(* CoDeSys 2.3 library: Visu_Scheduler_03_e.lib *)
(* Libraries: Standard.lib 4.10.05 11:14:46, SYSLIBCALLBACK.LIB*7.9.10 14:37:47 *)

(* POU Fu_Version_Visu_Scheduler, ST *)
FUNCTION Fu_Version_Visu_Scheduler : WORD
(*******************************************************************************
  WAGO Kontakttechnik GmbH Hansastr. 27 32423 Minden(Westf.) 
  Tel. +49571/887-0                                                                                                
   
  Function	: This function ist for checking purposes of the version.
 
  Version	: 3.1
  Date		: 14.03.2011

*******************************************************************************)
VAR_INPUT
	EN : BOOL;
END_VAR
Fu_Version_Visu_Scheduler:=16#0301;
(*
***** 26.01.2011, V3.0 *****************************************************
 - Release of the library Scheduler_03.lib and Visu_Scheduler_03.lib

***** 14.03.2011, V3.1*****************************************************
 - visuTimetable_e: Adjust the Input field for individual end time on Friday
*)
END_FUNCTION

(* Visualisation visuHoliday
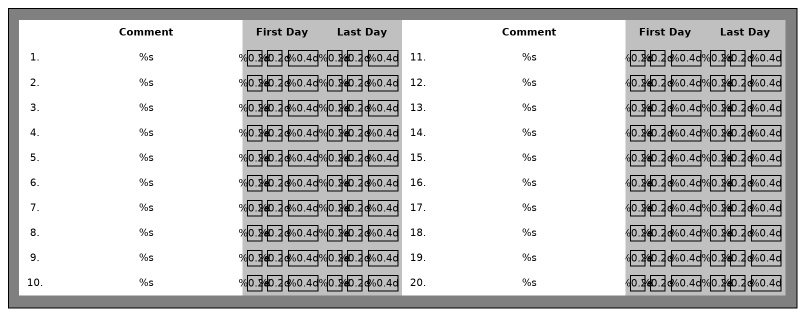
rectangle at (234,36)-(314,62): text "-     -"; tooltip First day Input format: DD-HH-YYYY
rectangle at (314,36)-(394,62): text "-     -"; tooltip Last day Input format: DD-HH-YYYY
rectangle at (319,42)-(334,58): text "%0.2d"; shows $typHoliday$.wLastDay[1,1]; editable 0..31
rectangle at (339,42)-(354,58): text "%0.2d"; shows $typHoliday$.wLastDay[2,1]; editable 0..12
rectangle at (360,42)-(390,58): text "%0.4d"; shows $typHoliday$.wLastDay[3,1]; editable 0..2099
rectangle at (43,36)-(234,62): text "%s"; shows $typHoliday$.strComment[1]; editable
rectangle at (234,62)-(314,87): text "-     -"; tooltip First day Input format: DD-HH-YYYY
rectangle at (314,62)-(394,87): text "-     -"; tooltip Last day Input format: DD-HH-YYYY
rectangle at (319,67)-(334,83): text "%0.2d"; shows $typHoliday$.wLastDay[1,2]; editable 0..31
rectangle at (339,67)-(354,83): text "%0.2d"; shows $typHoliday$.wLastDay[2,2]; editable 0..12
rectangle at (360,67)-(390,83): text "%0.4d"; shows $typHoliday$.wLastDay[3,2]; editable 0..2099
rectangle at (43,62)-(234,87): text "%s"; shows $typHoliday$.strComment[2]; editable
rectangle at (234,87)-(314,112): text "-     -"; tooltip First day Input format: DD-HH-YYYY
rectangle at (314,87)-(394,112): text "-     -"; tooltip Last day Input format: DD-HH-YYYY
rectangle at (319,92)-(334,108): text "%0.2d"; shows $typHoliday$.wLastDay[1,3]; editable 0..31
rectangle at (339,92)-(354,108): text "%0.2d"; shows $typHoliday$.wLastDay[2,3]; editable 0..12
rectangle at (360,92)-(390,108): text "%0.4d"; shows $typHoliday$.wLastDay[3,3]; editable 0..2099
rectangle at (43,87)-(234,112): text "%s"; shows $typHoliday$.strComment[3]; editable
rectangle at (234,112)-(314,137): text "-     -"; tooltip First day Input format: DD-HH-YYYY
rectangle at (314,112)-(394,137): text "-     -"; tooltip Last day Input format: DD-HH-YYYY
rectangle at (319,117)-(334,133): text "%0.2d"; shows $typHoliday$.wLastDay[1,4]; editable 0..31
rectangle at (339,117)-(354,133): text "%0.2d"; shows $typHoliday$.wLastDay[2,4]; editable 0..12
rectangle at (360,117)-(390,133): text "%0.4d"; shows $typHoliday$.wLastDay[3,4]; editable 0..2099
rectangle at (43,112)-(234,137): text "%s"; shows $typHoliday$.strComment[4]; editable
rectangle at (234,137)-(314,162): text "-     -"; tooltip First day Input format: DD-HH-YYYY
rectangle at (314,137)-(394,162): text "-     -"; tooltip Last day Input format: DD-HH-YYYY
rectangle at (319,142)-(334,158): text "%0.2d"; shows $typHoliday$.wLastDay[1,5]; editable 0..31
rectangle at (339,142)-(354,158): text "%0.2d"; shows $typHoliday$.wLastDay[2,5]; editable 0..12
rectangle at (360,142)-(390,158): text "%0.4d"; shows $typHoliday$.wLastDay[3,5]; editable 0..2099
rectangle at (43,137)-(234,162): text "%s"; shows $typHoliday$.strComment[5]; editable
rectangle at (234,162)-(314,187): text "-     -"; tooltip First day Input format: DD-HH-YYYY
rectangle at (314,162)-(394,187): text "-     -"; tooltip Last day Input format: DD-HH-YYYY
rectangle at (319,167)-(334,183): text "%0.2d"; shows $typHoliday$.wLastDay[1,6]; editable 0..31
rectangle at (339,167)-(354,183): text "%0.2d"; shows $typHoliday$.wLastDay[2,6]; editable 0..12
rectangle at (360,167)-(390,183): text "%0.4d"; shows $typHoliday$.wLastDay[3,6]; editable 0..2099
rectangle at (43,162)-(234,187): text "%s"; shows $typHoliday$.strComment[6]; editable
rectangle at (234,187)-(314,212): text "-     -"; tooltip First day Input format: DD-HH-YYYY
rectangle at (314,187)-(394,212): text "-     -"; tooltip Last day Input format: DD-HH-YYYY
rectangle at (319,192)-(334,208): text "%0.2d"; shows $typHoliday$.wLastDay[1,7]; editable 0..31
rectangle at (339,192)-(354,208): text "%0.2d"; shows $typHoliday$.wLastDay[2,7]; editable 0..12
rectangle at (360,192)-(390,208): text "%0.4d"; shows $typHoliday$.wLastDay[3,7]; editable 0..2099
rectangle at (43,187)-(234,212): text "%s"; shows $typHoliday$.strComment[7]; editable
rectangle at (234,212)-(314,237): text "-     -"; tooltip First day Input format: DD-HH-YYYY
rectangle at (314,212)-(394,237): text "-     -"; tooltip Last day Input format: DD-HH-YYYY
rectangle at (319,217)-(334,233): text "%0.2d"; shows $typHoliday$.wLastDay[1,8]; editable 0..31
rectangle at (339,217)-(354,233): text "%0.2d"; shows $typHoliday$.wLastDay[2,8]; editable 0..12
rectangle at (360,217)-(390,233): text "%0.4d"; shows $typHoliday$.wLastDay[3,8]; editable 0..2099
rectangle at (43,212)-(234,237): text "%s"; shows $typHoliday$.strComment[8]; editable
rectangle at (234,237)-(314,262): text "-     -"; tooltip First day Input format: DD-HH-YYYY
rectangle at (314,237)-(394,262): text "-     -"; tooltip Last day Input format: DD-HH-YYYY
rectangle at (319,242)-(334,258): text "%0.2d"; shows $typHoliday$.wLastDay[1,9]; editable 0..31
rectangle at (339,242)-(354,258): text "%0.2d"; shows $typHoliday$.wLastDay[2,9]; editable 0..12
rectangle at (360,242)-(390,258): text "%0.4d"; shows $typHoliday$.wLastDay[3,9]; editable 0..2099
rectangle at (43,237)-(234,262): text "%s"; shows $typHoliday$.strComment[9]; editable
rectangle at (234,262)-(314,287): text "-     -"; tooltip First day Input format: DD-HH-YYYY
rectangle at (314,262)-(394,287): text "-     -"; tooltip Last day Input format: DD-HH-YYYY
rectangle at (319,267)-(334,283): text "%0.2d"; shows $typHoliday$.wLastDay[1,10]; editable 0..31
rectangle at (339,267)-(354,283): text "%0.2d"; shows $typHoliday$.wLastDay[2,10]; editable 0..12
rectangle at (360,267)-(390,283): text "%0.4d"; shows $typHoliday$.wLastDay[3,10]; editable 0..2099
rectangle at (43,262)-(234,287): text "%s"; shows $typHoliday$.strComment[10]; editable
rectangle at (617,36)-(697,62): text "-     -"; tooltip First day Input format: DD-HH-YYYY
rectangle at (622,42)-(637,58): text "%0.2d"; shows $typHoliday$.wFirstDay[1,11]; editable 0..31
rectangle at (642,42)-(657,58): text "%0.2d"; shows $typHoliday$.wFirstDay[2,11]; editable 0..12
rectangle at (663,42)-(693,58): text "%0.4d"; shows $typHoliday$.wFirstDay[3,11]; editable 0..2099
rectangle at (697,36)-(777,62): text "-     -"; tooltip Last day Input format: DD-HH-YYYY
rectangle at (702,42)-(717,58): text "%0.2d"; shows $typHoliday$.wLastDay[1,11]; editable 0..31
rectangle at (722,42)-(737,58): text "%0.2d"; shows $typHoliday$.wLastDay[2,11]; editable 0..12
rectangle at (743,42)-(773,58): text "%0.4d"; shows $typHoliday$.wLastDay[3,11]; editable 0..2099
rectangle at (426,36)-(617,62): text "%s"; shows $typHoliday$.strComment[11]; editable
rectangle at (617,62)-(697,87): text "-     -"; tooltip First day Input format: DD-HH-YYYY
rectangle at (622,67)-(637,83): text "%0.2d"; shows $typHoliday$.wFirstDay[1,12]; editable 0..31
rectangle at (642,67)-(657,83): text "%0.2d"; shows $typHoliday$.wFirstDay[2,12]; editable 0..12
rectangle at (663,67)-(693,83): text "%0.4d"; shows $typHoliday$.wFirstDay[3,12]; editable 0..2099
rectangle at (697,62)-(777,87): text "-     -"; tooltip Last day Input format: DD-HH-YYYY
rectangle at (702,67)-(717,83): text "%0.2d"; shows $typHoliday$.wLastDay[1,12]; editable 0..31
rectangle at (722,67)-(737,83): text "%0.2d"; shows $typHoliday$.wLastDay[2,12]; editable 0..12
rectangle at (743,67)-(773,83): text "%0.4d"; shows $typHoliday$.wLastDay[3,12]; editable 0..2099
rectangle at (426,62)-(617,87): text "%s"; shows $typHoliday$.strComment[12]; editable
rectangle at (617,87)-(697,112): text "-     -"; tooltip First day Input format: DD-HH-YYYY
rectangle at (622,92)-(637,108): text "%0.2d"; shows $typHoliday$.wFirstDay[1,13]; editable 0..31
rectangle at (642,92)-(657,108): text "%0.2d"; shows $typHoliday$.wFirstDay[2,13]; editable 0..12
rectangle at (663,92)-(693,108): text "%0.4d"; shows $typHoliday$.wFirstDay[3,13]; editable 0..2099
rectangle at (697,87)-(777,112): text "-     -"; tooltip Last day Input format: DD-HH-YYYY
rectangle at (702,92)-(717,108): text "%0.2d"; shows $typHoliday$.wLastDay[1,13]; editable 0..31
rectangle at (722,92)-(737,108): text "%0.2d"; shows $typHoliday$.wLastDay[2,13]; editable 0..12
rectangle at (743,92)-(773,108): text "%0.4d"; shows $typHoliday$.wLastDay[3,13]; editable 0..2099
rectangle at (426,87)-(617,112): text "%s"; shows $typHoliday$.strComment[13]; editable
rectangle at (617,112)-(697,137): text "-     -"; tooltip First day Input format: DD-HH-YYYY
rectangle at (622,117)-(637,133): text "%0.2d"; shows $typHoliday$.wFirstDay[1,14]; editable 0..31
rectangle at (642,117)-(657,133): text "%0.2d"; shows $typHoliday$.wFirstDay[2,14]; editable 0..12
rectangle at (663,117)-(693,133): text "%0.4d"; shows $typHoliday$.wFirstDay[3,14]; editable 0..2099
rectangle at (697,112)-(777,137): text "-     -"; tooltip Last day Input format: DD-HH-YYYY
rectangle at (702,117)-(717,133): text "%0.2d"; shows $typHoliday$.wLastDay[1,14]; editable 0..31
rectangle at (722,117)-(737,133): text "%0.2d"; shows $typHoliday$.wLastDay[2,14]; editable 0..12
rectangle at (743,117)-(773,133): text "%0.4d"; shows $typHoliday$.wLastDay[3,14]; editable 0..2099
rectangle at (426,112)-(617,137): text "%s"; shows $typHoliday$.strComment[14]; editable
rectangle at (617,137)-(697,162): text "-     -"; tooltip First day Input format: DD-HH-YYYY
rectangle at (622,142)-(637,158): text "%0.2d"; shows $typHoliday$.wFirstDay[1,15]; editable 0..31
rectangle at (642,142)-(657,158): text "%0.2d"; shows $typHoliday$.wFirstDay[2,15]; editable 0..12
rectangle at (663,142)-(693,158): text "%0.4d"; shows $typHoliday$.wFirstDay[3,15]; editable 0..2099
rectangle at (697,137)-(777,162): text "-     -"; tooltip Last day Input format: DD-HH-YYYY
rectangle at (702,142)-(717,158): text "%0.2d"; shows $typHoliday$.wLastDay[1,15]; editable 0..31
rectangle at (722,142)-(737,158): text "%0.2d"; shows $typHoliday$.wLastDay[2,15]; editable 0..12
rectangle at (743,142)-(773,158): text "%0.4d"; shows $typHoliday$.wLastDay[3,15]; editable 0..2099
rectangle at (426,137)-(617,162): text "%s"; shows $typHoliday$.strComment[15]; editable
rectangle at (617,162)-(697,187): text "-     -"; tooltip First day Input format: DD-HH-YYYY
rectangle at (622,167)-(637,183): text "%0.2d"; shows $typHoliday$.wFirstDay[1,16]; editable 0..31
rectangle at (642,167)-(657,183): text "%0.2d"; shows $typHoliday$.wFirstDay[2,16]; editable 0..12
rectangle at (663,167)-(693,183): text "%0.4d"; shows $typHoliday$.wFirstDay[3,16]; editable 0..2099
rectangle at (697,162)-(777,187): text "-     -"; tooltip Last day Input format: DD-HH-YYYY
rectangle at (702,167)-(717,183): text "%0.2d"; shows $typHoliday$.wLastDay[1,16]; editable 0..31
rectangle at (722,167)-(737,183): text "%0.2d"; shows $typHoliday$.wLastDay[2,16]; editable 0..12
rectangle at (743,167)-(773,183): text "%0.4d"; shows $typHoliday$.wLastDay[3,16]; editable 0..2099
rectangle at (426,162)-(617,187): text "%s"; shows $typHoliday$.strComment[16]; editable
rectangle at (617,187)-(697,212): text "-     -"; tooltip First day Input format: DD-HH-YYYY
rectangle at (622,192)-(637,208): text "%0.2d"; shows $typHoliday$.wFirstDay[1,17]; editable 0..31
rectangle at (642,192)-(657,208): text "%0.2d"; shows $typHoliday$.wFirstDay[2,17]; editable 0..12
rectangle at (663,192)-(693,208): text "%0.4d"; shows $typHoliday$.wFirstDay[3,17]; editable 0..2099
rectangle at (697,187)-(777,212): text "-     -"; tooltip Last day Input format: DD-HH-YYYY
rectangle at (702,192)-(717,208): text "%0.2d"; shows $typHoliday$.wLastDay[1,17]; editable 0..31
rectangle at (722,192)-(737,208): text "%0.2d"; shows $typHoliday$.wLastDay[2,17]; editable 0..12
rectangle at (743,192)-(773,208): text "%0.4d"; shows $typHoliday$.wLastDay[3,17]; editable 0..2099
rectangle at (426,187)-(617,212): text "%s"; shows $typHoliday$.strComment[17]; editable
rectangle at (617,212)-(697,237): text "-     -"; tooltip First day Input format: DD-HH-YYYY
rectangle at (622,217)-(637,233): text "%0.2d"; shows $typHoliday$.wFirstDay[1,18]; editable 0..31
rectangle at (642,217)-(657,233): text "%0.2d"; shows $typHoliday$.wFirstDay[2,18]; editable 0..12
rectangle at (663,217)-(693,233): text "%0.4d"; shows $typHoliday$.wFirstDay[3,18]; editable 0..2099
rectangle at (697,212)-(777,237): text "-     -"; tooltip Last day Input format: DD-HH-YYYY
rectangle at (702,217)-(717,233): text "%0.2d"; shows $typHoliday$.wLastDay[1,18]; editable 0..31
rectangle at (722,217)-(737,233): text "%0.2d"; shows $typHoliday$.wLastDay[2,18]; editable 0..12
rectangle at (743,217)-(773,233): text "%0.4d"; shows $typHoliday$.wLastDay[3,18]; editable 0..2099
rectangle at (426,212)-(617,237): text "%s"; shows $typHoliday$.strComment[18]; editable
rectangle at (617,237)-(697,262): text "-     -"; tooltip First day Input format: DD-HH-YYYY
rectangle at (622,242)-(637,258): text "%0.2d"; shows $typHoliday$.wFirstDay[1,19]; editable 0..31
rectangle at (642,242)-(657,258): text "%0.2d"; shows $typHoliday$.wFirstDay[2,19]; editable 0..12
rectangle at (663,242)-(693,258): text "%0.4d"; shows $typHoliday$.wFirstDay[3,19]; editable 0..2099
rectangle at (697,237)-(777,262): text "-     -"; tooltip Last day Input format: DD-HH-YYYY
rectangle at (702,242)-(717,258): text "%0.2d"; shows $typHoliday$.wLastDay[1,19]; editable 0..31
rectangle at (722,242)-(737,258): text "%0.2d"; shows $typHoliday$.wLastDay[2,19]; editable 0..12
rectangle at (743,242)-(773,258): text "%0.4d"; shows $typHoliday$.wLastDay[3,19]; editable 0..2099
rectangle at (426,237)-(617,262): text "%s"; shows $typHoliday$.strComment[19]; editable
rectangle at (617,262)-(697,287): text "-     -"; tooltip First day Input format: DD-HH-YYYY
rectangle at (622,267)-(637,283): text "%0.2d"; shows $typHoliday$.wFirstDay[1,20]; editable 0..31
rectangle at (642,267)-(657,283): text "%0.2d"; shows $typHoliday$.wFirstDay[2,20]; editable 0..12
rectangle at (663,267)-(693,283): text "%0.4d"; shows $typHoliday$.wFirstDay[3,20]; editable 0..2099
rectangle at (697,262)-(777,287): text "-     -"; tooltip Last day Input format: DD-HH-YYYY
rectangle at (702,267)-(717,283): text "%0.2d"; shows $typHoliday$.wLastDay[1,20]; editable 0..31
rectangle at (722,267)-(737,283): text "%0.2d"; shows $typHoliday$.wLastDay[2,20]; editable 0..12
rectangle at (743,267)-(773,283): text "%0.4d"; shows $typHoliday$.wLastDay[3,20]; editable 0..2099
rectangle at (426,262)-(617,287): text "%s"; shows $typHoliday$.strComment[20]; editable
rectangle at (11,36)-(43,62): text "1."
rectangle at (11,62)-(43,87): text "2."
rectangle at (11,87)-(43,112): text "3."
rectangle at (11,112)-(43,137): text "4."
rectangle at (11,137)-(43,162): text "5."
rectangle at (11,162)-(43,187): text "6."
rectangle at (11,187)-(43,212): text "7."
rectangle at (11,212)-(43,237): text "8."
rectangle at (11,237)-(43,262): text "9."
rectangle at (11,262)-(43,287): text "10."
rectangle at (394,36)-(426,62): text "11."
rectangle at (394,62)-(426,87): text "12."
rectangle at (394,87)-(426,112): text "13."
rectangle at (394,112)-(426,137): text "14."
rectangle at (394,137)-(426,162): text "15."
rectangle at (394,162)-(426,187): text "16."
rectangle at (394,187)-(426,212): text "17."
rectangle at (394,212)-(426,237): text "18."
rectangle at (394,237)-(426,262): text "19."
rectangle at (394,262)-(426,287): text "20."
rectangle at (617,12)-(697,36): text "First Day"
rectangle at (697,12)-(777,36): text "Last Day"
rectangle at (426,12)-(617,36): text "Comment"
rectangle at (234,12)-(314,36): text "First Day"
rectangle at (314,12)-(394,36): text "Last Day"
rectangle at (43,12)-(234,36): text "Comment"
rectangle at (239,42)-(254,58): text "%0.2d"; shows $typHoliday$.wFirstDay[1,1]; editable 0..31
rectangle at (259,42)-(274,58): text "%0.2d"; shows $typHoliday$.wFirstDay[2,1]; editable 0..12
rectangle at (280,42)-(310,58): text "%0.4d"; shows $typHoliday$.wFirstDay[3,1]; editable 0..2099
rectangle at (239,67)-(254,83): text "%0.2d"; shows $typHoliday$.wFirstDay[1,2]; editable 0..31
rectangle at (259,67)-(274,83): text "%0.2d"; shows $typHoliday$.wFirstDay[2,2]; editable 0..12
rectangle at (280,67)-(310,83): text "%0.4d"; shows $typHoliday$.wFirstDay[3,2]; editable 0..2099
rectangle at (239,92)-(254,108): text "%0.2d"; shows $typHoliday$.wFirstDay[1,3]; editable 0..31
rectangle at (259,92)-(274,108): text "%0.2d"; shows $typHoliday$.wFirstDay[2,3]; editable 0..12
rectangle at (280,92)-(310,108): text "%0.4d"; shows $typHoliday$.wFirstDay[3,3]; editable 0..2099
rectangle at (239,117)-(254,133): text "%0.2d"; shows $typHoliday$.wFirstDay[1,4]; editable 0..31
rectangle at (259,117)-(274,133): text "%0.2d"; shows $typHoliday$.wFirstDay[2,4]; editable 0..12
rectangle at (280,117)-(310,133): text "%0.4d"; shows $typHoliday$.wFirstDay[3,4]; editable 0..2099
rectangle at (239,142)-(254,158): text "%0.2d"; shows $typHoliday$.wFirstDay[1,5]; editable 0..31
rectangle at (259,142)-(274,158): text "%0.2d"; shows $typHoliday$.wFirstDay[2,5]; editable 0..12
rectangle at (280,142)-(310,158): text "%0.4d"; shows $typHoliday$.wFirstDay[3,5]; editable 0..2099
rectangle at (239,167)-(254,183): text "%0.2d"; shows $typHoliday$.wFirstDay[1,6]; editable 0..31
rectangle at (259,167)-(274,183): text "%0.2d"; shows $typHoliday$.wFirstDay[2,6]; editable 0..12
rectangle at (280,167)-(310,183): text "%0.4d"; shows $typHoliday$.wFirstDay[3,6]; editable 0..2099
rectangle at (239,192)-(254,208): text "%0.2d"; shows $typHoliday$.wFirstDay[1,7]; editable 0..31
rectangle at (259,192)-(274,208): text "%0.2d"; shows $typHoliday$.wFirstDay[2,7]; editable 0..12
rectangle at (280,192)-(310,208): text "%0.4d"; shows $typHoliday$.wFirstDay[3,7]; editable 0..2099
rectangle at (239,217)-(254,233): text "%0.2d"; shows $typHoliday$.wFirstDay[1,8]; editable 0..31
rectangle at (259,217)-(274,233): text "%0.2d"; shows $typHoliday$.wFirstDay[2,8]; editable 0..12
rectangle at (280,217)-(310,233): text "%0.4d"; shows $typHoliday$.wFirstDay[3,8]; editable 0..2099
rectangle at (239,242)-(254,258): text "%0.2d"; shows $typHoliday$.wFirstDay[1,9]; editable 0..31
rectangle at (259,242)-(274,258): text "%0.2d"; shows $typHoliday$.wFirstDay[2,9]; editable 0..12
rectangle at (280,242)-(310,258): text "%0.4d"; shows $typHoliday$.wFirstDay[3,9]; editable 0..2099
rectangle at (239,267)-(254,283): text "%0.2d"; shows $typHoliday$.wFirstDay[1,10]; editable 0..31
rectangle at (259,267)-(274,283): text "%0.2d"; shows $typHoliday$.wFirstDay[2,10]; editable 0..12
rectangle at (280,267)-(310,283): text "%0.4d"; shows $typHoliday$.wFirstDay[3,10]; editable 0..2099
5 more shapes without text or variables
*)

(* Visualisation visuPublicHoliday
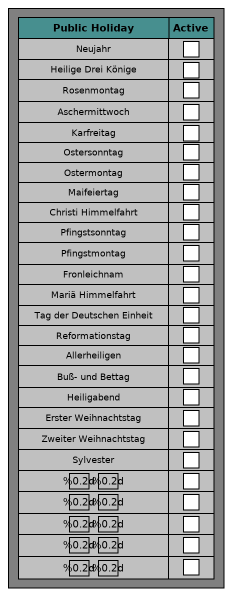
rectangle at (160,9)-(206,31): text "Active"
rectangle at (10,9)-(161,31): text "Public Holiday"
rectangle at (10,30)-(161,52): text "Neujahr"
rectangle at (175,33)-(191,49): alarm colour if $typPublicHoliday$.Neujahr; toggles $typPublicHoliday$.Neujahr; tooltip Wenn dieses Feld aktiviert ist, wird der Feiertag für die Feiertagserkennung im "FbPublicHoliday" berücksichtigt.
rectangle at (10,51)-(161,72): text "Heilige Drei Könige"
rectangle at (175,54)-(191,70): alarm colour if $typPublicHoliday$.Heilige_Drei_Koenige; toggles $typPublicHoliday$.Heilige_Drei_Koenige; tooltip Wenn dieses Feld aktiviert ist, wird der Feiertag für die Feiertagserkennung im "FbPublicHoliday" berücksichtigt.
rectangle at (10,71)-(161,94): text "Rosenmontag"
rectangle at (175,74)-(191,90): alarm colour if $typPublicHoliday$.Rosenmontag; toggles $typPublicHoliday$.Rosenmontag; tooltip Wenn dieses Feld aktiviert ist, wird der Feiertag für die Feiertagserkennung im "FbPublicHoliday" berücksichtigt.
rectangle at (10,93)-(161,115): text "Aschermittwoch"
rectangle at (175,96)-(191,112): alarm colour if $typPublicHoliday$.Aschermittwoch; toggles $typPublicHoliday$.Aschermittwoch; tooltip Wenn dieses Feld aktiviert ist, wird der Feiertag für die Feiertagserkennung im "FbPublicHoliday" berücksichtigt.
rectangle at (10,114)-(161,136): text "Karfreitag"
rectangle at (175,117)-(191,133): alarm colour if $typPublicHoliday$.Karfreitag; toggles $typPublicHoliday$.Karfreitag; tooltip Wenn dieses Feld aktiviert ist, wird der Feiertag für die Feiertagserkennung im "FbPublicHoliday" berücksichtigt.
rectangle at (10,134)-(161,155): text "Ostersonntag"
rectangle at (175,136)-(191,152): alarm colour if $typPublicHoliday$.Ostersonntag; toggles $typPublicHoliday$.Ostersonntag; tooltip Wenn dieses Feld aktiviert ist, wird der Feiertag für die Feiertagserkennung im "FbPublicHoliday" berücksichtigt.
rectangle at (10,154)-(161,176): text "Ostermontag"
rectangle at (175,156)-(191,172): alarm colour if $typPublicHoliday$.Ostermontag; toggles $typPublicHoliday$.Ostermontag; tooltip Wenn dieses Feld aktiviert ist, wird der Feiertag für die Feiertagserkennung im "FbPublicHoliday" berücksichtigt.
rectangle at (10,174)-(161,195): text "Maifeiertag"
rectangle at (175,176)-(191,192): alarm colour if $typPublicHoliday$.Maifeiertag; toggles $typPublicHoliday$.Maifeiertag; tooltip Wenn dieses Feld aktiviert ist, wird der Feiertag für die Feiertagserkennung im "FbPublicHoliday" berücksichtigt.
rectangle at (10,194)-(161,215): text "Christi Himmelfahrt"
rectangle at (175,196)-(191,212): alarm colour if $typPublicHoliday$.Christi_Himmelfahrt; toggles $typPublicHoliday$.Christi_Himmelfahrt; tooltip Wenn dieses Feld aktiviert ist, wird der Feiertag für die Feiertagserkennung im "FbPublicHoliday" berücksichtigt.
rectangle at (10,214)-(161,235): text "Pfingstsonntag"
rectangle at (175,216)-(191,232): alarm colour if $typPublicHoliday$.Pfingstsonntag; toggles $typPublicHoliday$.Pfingstsonntag; tooltip Wenn dieses Feld aktiviert ist, wird der Feiertag für die Feiertagserkennung im "FbPublicHoliday" berücksichtigt.
rectangle at (10,234)-(161,257): text "Pfingstmontag"
rectangle at (175,237)-(191,253): alarm colour if $typPublicHoliday$.Pfingstmontag; toggles $typPublicHoliday$.Pfingstmontag; tooltip Wenn dieses Feld aktiviert ist, wird der Feiertag für die Feiertagserkennung im "FbPublicHoliday" berücksichtigt.
rectangle at (10,256)-(161,277): text "Fronleichnam"
rectangle at (175,258)-(191,274): alarm colour if $typPublicHoliday$.Fronleichnam; toggles $typPublicHoliday$.Fronleichnam; tooltip Wenn dieses Feld aktiviert ist, wird der Feiertag für die Feiertagserkennung im "FbPublicHoliday" berücksichtigt.
rectangle at (10,276)-(161,298): text "Mariä Himmelfahrt"
rectangle at (175,279)-(191,295): alarm colour if $typPublicHoliday$.Mariae_Himmelfahrt; toggles $typPublicHoliday$.Mariae_Himmelfahrt; tooltip Wenn dieses Feld aktiviert ist, wird der Feiertag für die Feiertagserkennung im "FbPublicHoliday" berücksichtigt.
rectangle at (10,297)-(161,318): text "Tag der Deutschen Einheit"
rectangle at (175,299)-(191,315): alarm colour if $typPublicHoliday$.Tag_der_Deutschen_Einheit; toggles $typPublicHoliday$.Tag_der_Deutschen_Einheit; tooltip Wenn dieses Feld aktiviert ist, wird der Feiertag für die Feiertagserkennung im "FbPublicHoliday" berücksichtigt.
rectangle at (10,317)-(161,339): text "Reformationstag"
rectangle at (175,319)-(191,335): alarm colour if $typPublicHoliday$.Reformationstag; toggles $typPublicHoliday$.Reformationstag; tooltip Wenn dieses Feld aktiviert ist, wird der Feiertag für die Feiertagserkennung im "FbPublicHoliday" berücksichtigt.
rectangle at (10,337)-(161,358): text "Allerheiligen"
rectangle at (175,339)-(191,355): alarm colour if $typPublicHoliday$.Allerheiligen; toggles $typPublicHoliday$.Allerheiligen; tooltip Wenn dieses Feld aktiviert ist, wird der Feiertag für die Feiertagserkennung im "FbPublicHoliday" berücksichtigt.
rectangle at (10,357)-(161,381): text "Buß- und Bettag"
rectangle at (175,360)-(191,376): alarm colour if $typPublicHoliday$.Buss_und_Bettag; toggles $typPublicHoliday$.Buss_und_Bettag; tooltip Wenn dieses Feld aktiviert ist, wird der Feiertag für die Feiertagserkennung im "FbPublicHoliday" berücksichtigt.
rectangle at (10,379)-(161,400): text "Heiligabend"
rectangle at (175,381)-(191,397): alarm colour if $typPublicHoliday$.Heiligabend; toggles $typPublicHoliday$.Heiligabend; tooltip Wenn dieses Feld aktiviert ist, wird der Feiertag für die Feiertagserkennung im "FbPublicHoliday" berücksichtigt.
rectangle at (10,399)-(161,421): text "Erster Weihnachtstag"
rectangle at (175,402)-(191,418): alarm colour if $typPublicHoliday$.Erster_Weihnachtstag; toggles $typPublicHoliday$.Erster_Weihnachtstag; tooltip Wenn dieses Feld aktiviert ist, wird der Feiertag für die Feiertagserkennung im "FbPublicHoliday" berücksichtigt.
rectangle at (10,420)-(161,442): text "Zweiter Weihnachtstag"
rectangle at (175,423)-(191,439): alarm colour if $typPublicHoliday$.Zweiter_Weihnachtstag; toggles $typPublicHoliday$.Zweiter_Weihnachtstag; tooltip Wenn dieses Feld aktiviert ist, wird der Feiertag für die Feiertagserkennung im "FbPublicHoliday" berücksichtigt.
rectangle at (10,441)-(161,463): text "Sylvester"
rectangle at (175,444)-(191,460): alarm colour if $typPublicHoliday$.Sylvester; toggles $typPublicHoliday$.Sylvester; tooltip Wenn dieses Feld aktiviert ist, wird der Feiertag für die Feiertagserkennung im "FbPublicHoliday" berücksichtigt.
rectangle at (10,462)-(161,485): text "-"; tooltip Eingabeformat:DD-MM Es können beliebige Feiertage mit ihrem Datum vorgegeben werden.
rectangle at (175,465)-(191,481): alarm colour if $typPublicHoliday$.SetSpecialPublicHoliday.0; toggles $typPublicHoliday$.SetSpecialPublicHoliday.0; tooltip Wenn dieses Feld aktiviert ist, wird der Feiertag für die Feiertagserkennung im "FbPublicHoliday" berücksichtigt.
rectangle at (10,483)-(161,506): text "-"; tooltip Eingabeformat:DD-MM Es können beliebige Feiertage mit ihrem Datum vorgegeben werden.
rectangle at (10,505)-(161,528): text "-"; tooltip Eingabeformat:DD-MM Es können beliebige Feiertage mit ihrem Datum vorgegeben werden.
rectangle at (10,526)-(161,549): text "-"; tooltip Eingabeformat:DD-MM Es können beliebige Feiertage mit ihrem Datum vorgegeben werden.
rectangle at (10,548)-(161,571): text "-"; tooltip Eingabeformat:DD-MM Es können beliebige Feiertage mit ihrem Datum vorgegeben werden.
rectangle at (175,486)-(191,502): alarm colour if $typPublicHoliday$.SetSpecialPublicHoliday.1; toggles $typPublicHoliday$.SetSpecialPublicHoliday.1; tooltip Wenn dieses Feld aktiviert ist, wird der Feiertag für die Feiertagserkennung im "FbPublicHoliday" berücksichtigt.
rectangle at (175,508)-(191,524): alarm colour if $typPublicHoliday$.SetSpecialPublicHoliday.2; toggles $typPublicHoliday$.SetSpecialPublicHoliday.2; tooltip Wenn dieses Feld aktiviert ist, wird der Feiertag für die Feiertagserkennung im "FbPublicHoliday" berücksichtigt.
rectangle at (175,529)-(191,545): alarm colour if $typPublicHoliday$.SetSpecialPublicHoliday.3; toggles $typPublicHoliday$.SetSpecialPublicHoliday.3; tooltip Wenn dieses Feld aktiviert ist, wird der Feiertag für die Feiertagserkennung im "FbPublicHoliday" berücksichtigt.
rectangle at (175,551)-(191,567): alarm colour if $typPublicHoliday$.SetSpecialPublicHoliday.4; toggles $typPublicHoliday$.SetSpecialPublicHoliday.4; tooltip Wenn dieses Feld aktiviert ist, wird der Feiertag für die Feiertagserkennung im "FbPublicHoliday" berücksichtigt.
rectangle at (90,465)-(110,481): text "%0.2d"; shows $typPublicHoliday$.SpecialPublicHoliday1_month; editable 1..12
rectangle at (61,465)-(81,481): text "%0.2d"; shows $typPublicHoliday$.SpecialPublicHoliday1_day; editable 1..31
rectangle at (90,486)-(110,502): text "%0.2d"; shows $typPublicHoliday$.SpecialPublicHoliday2_month; editable 1..12
rectangle at (61,486)-(81,502): text "%0.2d"; shows $typPublicHoliday$.SpecialPublicHoliday2_day; editable 1..31
rectangle at (90,508)-(110,524): text "%0.2d"; shows $typPublicHoliday$.SpecialPublicHoliday3_month; editable 1..12
rectangle at (61,508)-(81,524): text "%0.2d"; shows $typPublicHoliday$.SpecialPublicHoliday3_day; editable 1..31
rectangle at (90,529)-(110,545): text "%0.2d"; shows $typPublicHoliday$.SpecialPublicHoliday4_month; editable 1..12
rectangle at (61,529)-(81,545): text "%0.2d"; shows $typPublicHoliday$.SpecialPublicHoliday4_day; editable 1..31
rectangle at (90,552)-(110,568): text "%0.2d"; shows $typPublicHoliday$.SpecialPublicHoliday5_month; editable 1..12
rectangle at (61,552)-(81,568): text "%0.2d"; shows $typPublicHoliday$.SpecialPublicHoliday5_day; editable 1..31
27 more shapes without text or variables
*)

(* Visualisation visuScheduler_HolidayParty
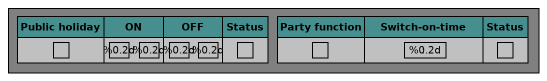
rectangle at (95,8)-(156,30): text "ON"
rectangle at (155,8)-(215,30): text "OFF"
rectangle at (474,8)-(520,30): text "Status"
rectangle at (489,34)-(505,50): alarm colour if $typSchedule$.Party_active.0; tooltip Indicates if time condition is fulfilled
rectangle at (95,29)-(156,55): text ":"; tooltip Switch ON time of the public holiday
rectangle at (101,34)-(121,50): text "%0.2d"; shows $typSchedule$.PublicHolidayON_hour; editable 0..24
rectangle at (131,34)-(151,50): text "%0.2d"; shows $typSchedule$.PublicHolidayON_minute; editable 0..59
rectangle at (155,29)-(215,55): text ":"; tooltip Switch OFF time of the public holiday
rectangle at (161,34)-(181,50): text "%0.2d"; shows $typSchedule$.PublicHolidayOff_hour; editable 0..24
rectangle at (190,34)-(210,50): text "%0.2d"; shows $typSchedule$.PublicHolidayOff_minute; editable 0..59
rectangle at (214,8)-(260,30): text "Status"
rectangle at (229,34)-(245,50): alarm colour if $typSchedule$.PublicHoliday_active.0; tooltip Indicates if time condition is fulfilled
rectangle at (269,8)-(357,30): text "Party function"
rectangle at (269,29)-(357,55): text ":"
rectangle at (304,34)-(320,50): alarm colour if $typSchedule$.StatusScheduler.4; tooltip Indicates if time condition is fulfilled
rectangle at (356,8)-(475,30): text "Switch-on-time"
rectangle at (356,29)-(475,55): text ":"
rectangle at (9,8)-(96,30): text "Public holiday"
rectangle at (45,34)-(61,50): alarm colour if $typSchedule$.StatusScheduler.3; tooltip Indicates if time condition is fulfilled
rectangle at (396,34)-(438,50): text "%0.2d"; shows $typSchedule$.Party_length; editable
4 more shapes without text or variables
*)

(* Visualisation visuScheduler_HolidayPartyValue
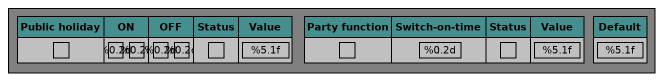
rectangle at (95,8)-(141,30): text "ON"
rectangle at (140,8)-(186,30): text "OFF"
rectangle at (477,8)-(523,30): text "Status"
rectangle at (492,34)-(508,50): alarm colour if $typSchedule$.Party_active.0; tooltip Indicates if time condition is fulfilled
rectangle at (95,29)-(141,55): text ":"; tooltip Switch ON time of the public holiday
rectangle at (100,34)-(115,50): text "%0.2d"; shows $typSchedule$.PublicHolidayON_hour; editable 0..24
rectangle at (121,34)-(136,50): text "%0.2d"; shows $typSchedule$.PublicHolidayON_minute; editable 0..59
rectangle at (140,29)-(186,55): text ":"; tooltip Switch OFF time of the public holiday
rectangle at (145,34)-(160,50): text "%0.2d"; shows $typSchedule$.PublicHolidayOff_hour; editable 0..24
rectangle at (166,34)-(181,50): text "%0.2d"; shows $typSchedule$.PublicHolidayOff_minute; editable 0..59
rectangle at (185,8)-(231,30): text "Status"
rectangle at (200,34)-(216,50): alarm colour if $typSchedule$.PublicHoliday_active.0; tooltip Indicates if time condition is fulfilled
rectangle at (296,8)-(384,30): text "Party function"
rectangle at (296,29)-(384,55): text ":"
rectangle at (331,34)-(347,50): alarm colour if $typSchedule$.StatusScheduler.4; tooltip Indicates if time condition is fulfilled
rectangle at (383,8)-(478,30): text "Switch-on-time"
rectangle at (383,29)-(478,55): text ":"
rectangle at (9,8)-(96,30): text "Public holiday"
rectangle at (45,34)-(61,50): alarm colour if $typSchedule$.StatusScheduler.3; tooltip Indicates if time condition is fulfilled
rectangle at (411,34)-(453,50): text "%0.2d"; shows $typSchedule$.Party_length; editable
rectangle at (230,8)-(284,30): text "Value"
rectangle at (230,29)-(284,55): tooltip Value of the scheduler Puplic holiday
rectangle at (234,34)-(281,50): text "%5.1f"; shows $typScheduleValue$.rHoliday; editable
rectangle at (522,8)-(576,30): text "Value"
rectangle at (522,29)-(576,55): tooltip Value of the scheduler Party function
rectangle at (526,34)-(572,50): text "%5.1f"; shows $typScheduleValue$.rParty; editable
rectangle at (585,8)-(639,30): text "Default"
rectangle at (585,29)-(639,55): tooltip Default-Value of the scheduler
rectangle at (589,34)-(635,50): text "%5.1f"; shows $typScheduleValue$.rDefault; editable
4 more shapes without text or variables
*)

(* Visualisation visuScheduler_SpecialPeriods
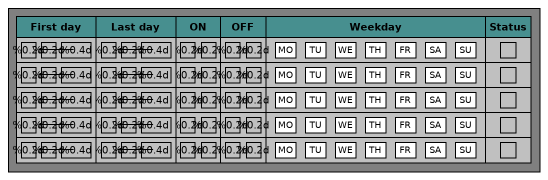
rectangle at (167,8)-(213,30): text "ON"
rectangle at (257,8)-(478,30): text "Weekday"
rectangle at (212,8)-(258,30): text "OFF"
rectangle at (87,8)-(168,30): text "Last day"
rectangle at (8,8)-(88,30): text "First day"
rectangle at (477,8)-(523,30): text "Status"
rectangle at (257,29)-(478,55): tooltip Activation of the days of the week when the scheduler should be enabled
rectangle at (267,34)-(288,50): text "MO"; alarm colour if $typSchedule$.ScheduleSpecialPeriods[1].Weekday.0; toggles $typSchedule$.ScheduleSpecialPeriods[1].Weekday.0
rectangle at (297,34)-(318,50): text "TU"; alarm colour if $typSchedule$.ScheduleSpecialPeriods[1].Weekday.1; toggles $typSchedule$.ScheduleSpecialPeriods[1].Weekday.1
rectangle at (327,34)-(348,50): text "WE"; alarm colour if $typSchedule$.ScheduleSpecialPeriods[1].Weekday.2; toggles $typSchedule$.ScheduleSpecialPeriods[1].Weekday.2
rectangle at (357,34)-(378,50): text "TH"; alarm colour if $typSchedule$.ScheduleSpecialPeriods[1].Weekday.3; toggles $typSchedule$.ScheduleSpecialPeriods[1].Weekday.3
rectangle at (387,34)-(408,50): text "FR"; alarm colour if $typSchedule$.ScheduleSpecialPeriods[1].Weekday.4; toggles $typSchedule$.ScheduleSpecialPeriods[1].Weekday.4
rectangle at (417,34)-(438,50): text "SA"; alarm colour if $typSchedule$.ScheduleSpecialPeriods[1].Weekday.5; toggles $typSchedule$.ScheduleSpecialPeriods[1].Weekday.5
rectangle at (447,34)-(468,50): text "SU"; alarm colour if $typSchedule$.ScheduleSpecialPeriods[1].Weekday.6; toggles $typSchedule$.ScheduleSpecialPeriods[1].Weekday.6
rectangle at (492,34)-(508,50): alarm colour if $typSchedule$.ScheduleSpecialPeriods[1].Active.0; tooltip Indicates if time condition is fulfilled
rectangle at (167,29)-(213,55): text ":"; tooltip Switch ON time of the scheduler single period
rectangle at (172,34)-(187,50): text "%0.2d"; shows $typSchedule$.ScheduleSpecialPeriods[1].ON_hour; editable 0..23
rectangle at (193,34)-(208,50): text "%0.2d"; shows $typSchedule$.ScheduleSpecialPeriods[1].ON_minute; editable 0..59
rectangle at (87,29)-(168,55): text "_______"; tooltip Last day of the scheduler single period Input format: DD-HH-YYYY
rectangle at (93,34)-(108,50): text "%0.2d"; shows $typSchedule$.ScheduleSpecialPeriods[1].LastDay_day; editable 1..31
rectangle at (113,34)-(128,50): text "%0.2d"; shows $typSchedule$.ScheduleSpecialPeriods[1].LastDay_month; editable 1..12
rectangle at (133,34)-(163,50): text "%0.4d"; shows $typSchedule$.ScheduleSpecialPeriods[1].LastDay_year; editable 0000..2100
rectangle at (8,29)-(88,55): text "_______"; tooltip First day of the scheduler single period Input format: DD-HH-YYYY
rectangle at (33,34)-(48,50): text "%0.2d"; shows $typSchedule$.ScheduleSpecialPeriods[1].FirstDay_month; editable 1..12
rectangle at (13,34)-(28,50): text "%0.2d"; shows $typSchedule$.ScheduleSpecialPeriods[1].FirstDay_day; editable 1..31
rectangle at (53,34)-(83,50): text "%0.4d"; shows $typSchedule$.ScheduleSpecialPeriods[1].FirstDay_year; editable 0000..2100
rectangle at (212,29)-(258,55): text ":"; tooltip Switch OFF time of the scheduler single period
rectangle at (217,34)-(232,50): text "%0.2d"; shows $typSchedule$.ScheduleSpecialPeriods[1].OFF_hour; editable 0..23
rectangle at (238,34)-(253,50): text "%0.2d"; shows $typSchedule$.ScheduleSpecialPeriods[1].OFF_minute; editable 0..59
rectangle at (257,54)-(478,80): tooltip Activation of the days of the week when the scheduler should be enabled
rectangle at (267,59)-(288,75): text "MO"; alarm colour if $typSchedule$.ScheduleSpecialPeriods[2].Weekday.0; toggles $typSchedule$.ScheduleSpecialPeriods[2].Weekday.0
rectangle at (297,59)-(318,75): text "TU"; alarm colour if $typSchedule$.ScheduleSpecialPeriods[2].Weekday.1; toggles $typSchedule$.ScheduleSpecialPeriods[2].Weekday.1
rectangle at (327,59)-(348,75): text "WE"; alarm colour if $typSchedule$.ScheduleSpecialPeriods[2].Weekday.2; toggles $typSchedule$.ScheduleSpecialPeriods[2].Weekday.2
rectangle at (357,59)-(378,75): text "TH"; alarm colour if $typSchedule$.ScheduleSpecialPeriods[2].Weekday.3; toggles $typSchedule$.ScheduleSpecialPeriods[2].Weekday.3
rectangle at (387,59)-(408,75): text "FR"; alarm colour if $typSchedule$.ScheduleSpecialPeriods[2].Weekday.4; toggles $typSchedule$.ScheduleSpecialPeriods[2].Weekday.4
rectangle at (417,59)-(438,75): text "SA"; alarm colour if $typSchedule$.ScheduleSpecialPeriods[2].Weekday.5; toggles $typSchedule$.ScheduleSpecialPeriods[2].Weekday.5
rectangle at (447,59)-(468,75): text "SU"; alarm colour if $typSchedule$.ScheduleSpecialPeriods[2].Weekday.6; toggles $typSchedule$.ScheduleSpecialPeriods[2].Weekday.6
rectangle at (492,59)-(508,75): alarm colour if $typSchedule$.ScheduleSpecialPeriods[2].Active.0; tooltip Indicates if time condition is fulfilled
rectangle at (167,54)-(213,80): text ":"; tooltip Switch ON time of the scheduler single period
rectangle at (172,59)-(187,75): text "%0.2d"; shows $typSchedule$.ScheduleSpecialPeriods[2].ON_hour; editable 0..23
rectangle at (193,59)-(208,75): text "%0.2d"; shows $typSchedule$.ScheduleSpecialPeriods[2].ON_minute; editable 0..59
rectangle at (87,54)-(168,80): text "_______"; tooltip Last day of the scheduler single period Input format: DD-HH-YYYY
rectangle at (93,59)-(108,75): text "%0.2d"; shows $typSchedule$.ScheduleSpecialPeriods[2].LastDay_day; editable 1..31
rectangle at (113,59)-(128,75): text "%0.2d"; shows $typSchedule$.ScheduleSpecialPeriods[2].LastDay_month; editable 1..12
rectangle at (133,59)-(163,75): text "%0.4d"; shows $typSchedule$.ScheduleSpecialPeriods[2].LastDay_year; editable 0000..2100
rectangle at (8,54)-(88,80): text "_______"; tooltip First day of the scheduler single period Input format: DD-HH-YYYY
rectangle at (33,59)-(48,75): text "%0.2d"; shows $typSchedule$.ScheduleSpecialPeriods[2].FirstDay_month; editable 1..12
rectangle at (13,59)-(28,75): text "%0.2d"; shows $typSchedule$.ScheduleSpecialPeriods[2].FirstDay_day; editable 1..31
rectangle at (53,59)-(83,75): text "%0.4d"; shows $typSchedule$.ScheduleSpecialPeriods[2].FirstDay_year; editable 0000..2100
rectangle at (212,54)-(258,80): text ":"; tooltip Switch OFF time of the scheduler single period
rectangle at (217,59)-(232,75): text "%0.2d"; shows $typSchedule$.ScheduleSpecialPeriods[2].OFF_hour; editable 0..23
rectangle at (238,59)-(253,75): text "%0.2d"; shows $typSchedule$.ScheduleSpecialPeriods[2].OFF_minute; editable 0..59
rectangle at (257,79)-(478,105): tooltip Activation of the days of the week when the scheduler should be enabled
rectangle at (267,84)-(288,100): text "MO"; alarm colour if $typSchedule$.ScheduleSpecialPeriods[3].Weekday.0; toggles $typSchedule$.ScheduleSpecialPeriods[3].Weekday.0
rectangle at (297,84)-(318,100): text "TU"; alarm colour if $typSchedule$.ScheduleSpecialPeriods[3].Weekday.1; toggles $typSchedule$.ScheduleSpecialPeriods[3].Weekday.1
rectangle at (327,84)-(348,100): text "WE"; alarm colour if $typSchedule$.ScheduleSpecialPeriods[3].Weekday.2; toggles $typSchedule$.ScheduleSpecialPeriods[3].Weekday.2
rectangle at (357,84)-(378,100): text "TH"; alarm colour if $typSchedule$.ScheduleSpecialPeriods[3].Weekday.3; toggles $typSchedule$.ScheduleSpecialPeriods[3].Weekday.3
rectangle at (387,84)-(408,100): text "FR"; alarm colour if $typSchedule$.ScheduleSpecialPeriods[3].Weekday.4; toggles $typSchedule$.ScheduleSpecialPeriods[3].Weekday.4
rectangle at (417,84)-(438,100): text "SA"; alarm colour if $typSchedule$.ScheduleSpecialPeriods[3].Weekday.5; toggles $typSchedule$.ScheduleSpecialPeriods[3].Weekday.5
rectangle at (447,84)-(468,100): text "SU"; alarm colour if $typSchedule$.ScheduleSpecialPeriods[3].Weekday.6; toggles $typSchedule$.ScheduleSpecialPeriods[3].Weekday.6
rectangle at (492,84)-(508,100): alarm colour if $typSchedule$.ScheduleSpecialPeriods[3].Active.0; tooltip Indicates if time condition is fulfilled
rectangle at (167,79)-(213,105): text ":"; tooltip Switch ON time of the scheduler single period
rectangle at (172,84)-(187,100): text "%0.2d"; shows $typSchedule$.ScheduleSpecialPeriods[3].ON_hour; editable 0..23
rectangle at (193,84)-(208,100): text "%0.2d"; shows $typSchedule$.ScheduleSpecialPeriods[3].ON_minute; editable 0..59
rectangle at (87,79)-(168,105): text "_______"; tooltip Last day of the scheduler single period Input format: DD-HH-YYYY
rectangle at (93,84)-(108,100): text "%0.2d"; shows $typSchedule$.ScheduleSpecialPeriods[3].LastDay_day; editable 1..31
rectangle at (113,84)-(128,100): text "%0.2d"; shows $typSchedule$.ScheduleSpecialPeriods[3].LastDay_month; editable 1..12
rectangle at (133,84)-(163,100): text "%0.4d"; shows $typSchedule$.ScheduleSpecialPeriods[3].LastDay_year; editable 0000..2100
rectangle at (8,79)-(88,105): text "_______"; tooltip First day of the scheduler single period Input format: DD-HH-YYYY
rectangle at (33,84)-(48,100): text "%0.2d"; shows $typSchedule$.ScheduleSpecialPeriods[3].FirstDay_month; editable 1..12
rectangle at (13,84)-(28,100): text "%0.2d"; shows $typSchedule$.ScheduleSpecialPeriods[3].FirstDay_day; editable 1..31
rectangle at (53,84)-(83,100): text "%0.4d"; shows $typSchedule$.ScheduleSpecialPeriods[3].FirstDay_year; editable 0000..2100
rectangle at (212,79)-(258,105): text ":"; tooltip Switch OFF time of the scheduler single period
rectangle at (217,84)-(232,100): text "%0.2d"; shows $typSchedule$.ScheduleSpecialPeriods[3].OFF_hour; editable 0..23
rectangle at (238,84)-(253,100): text "%0.2d"; shows $typSchedule$.ScheduleSpecialPeriods[3].OFF_minute; editable 0..59
rectangle at (257,104)-(478,130): tooltip Activation of the days of the week when the scheduler should be enabled
rectangle at (267,109)-(288,125): text "MO"; alarm colour if $typSchedule$.ScheduleSpecialPeriods[4].Weekday.0; toggles $typSchedule$.ScheduleSpecialPeriods[4].Weekday.0
rectangle at (297,109)-(318,125): text "TU"; alarm colour if $typSchedule$.ScheduleSpecialPeriods[4].Weekday.1; toggles $typSchedule$.ScheduleSpecialPeriods[4].Weekday.1
rectangle at (327,109)-(348,125): text "WE"; alarm colour if $typSchedule$.ScheduleSpecialPeriods[4].Weekday.2; toggles $typSchedule$.ScheduleSpecialPeriods[4].Weekday.2
rectangle at (357,109)-(378,125): text "TH"; alarm colour if $typSchedule$.ScheduleSpecialPeriods[4].Weekday.3; toggles $typSchedule$.ScheduleSpecialPeriods[4].Weekday.3
rectangle at (387,109)-(408,125): text "FR"; alarm colour if $typSchedule$.ScheduleSpecialPeriods[4].Weekday.4; toggles $typSchedule$.ScheduleSpecialPeriods[4].Weekday.4
rectangle at (417,109)-(438,125): text "SA"; alarm colour if $typSchedule$.ScheduleSpecialPeriods[4].Weekday.5; toggles $typSchedule$.ScheduleSpecialPeriods[4].Weekday.5
rectangle at (447,109)-(468,125): text "SU"; alarm colour if $typSchedule$.ScheduleSpecialPeriods[4].Weekday.6; toggles $typSchedule$.ScheduleSpecialPeriods[4].Weekday.6
rectangle at (492,109)-(508,125): alarm colour if $typSchedule$.ScheduleSpecialPeriods[4].Active.0; tooltip Indicates if time condition is fulfilled
rectangle at (167,104)-(213,130): text ":"; tooltip Switch ON time of the scheduler single period
rectangle at (172,109)-(187,125): text "%0.2d"; shows $typSchedule$.ScheduleSpecialPeriods[4].ON_hour; editable 0..23
rectangle at (193,109)-(208,125): text "%0.2d"; shows $typSchedule$.ScheduleSpecialPeriods[4].ON_minute; editable 0..59
rectangle at (87,104)-(168,130): text "_______"; tooltip Last day of the scheduler single period Input format: DD-HH-YYYY
rectangle at (93,109)-(108,125): text "%0.2d"; shows $typSchedule$.ScheduleSpecialPeriods[4].LastDay_day; editable 1..31
rectangle at (113,109)-(128,125): text "%0.2d"; shows $typSchedule$.ScheduleSpecialPeriods[4].LastDay_month; editable 1..12
rectangle at (133,109)-(163,125): text "%0.4d"; shows $typSchedule$.ScheduleSpecialPeriods[4].LastDay_year; editable 0000..2100
rectangle at (8,104)-(88,130): text "_______"; tooltip First day of the scheduler single period Input format: DD-HH-YYYY
rectangle at (33,109)-(48,125): text "%0.2d"; shows $typSchedule$.ScheduleSpecialPeriods[4].FirstDay_month; editable 1..12
rectangle at (13,109)-(28,125): text "%0.2d"; shows $typSchedule$.ScheduleSpecialPeriods[4].FirstDay_day; editable 1..31
rectangle at (53,109)-(83,125): text "%0.4d"; shows $typSchedule$.ScheduleSpecialPeriods[4].FirstDay_year; editable 0000..2100
rectangle at (212,104)-(258,130): text ":"; tooltip Switch OFF time of the scheduler single period
rectangle at (217,109)-(232,125): text "%0.2d"; shows $typSchedule$.ScheduleSpecialPeriods[4].OFF_hour; editable 0..23
rectangle at (238,109)-(253,125): text "%0.2d"; shows $typSchedule$.ScheduleSpecialPeriods[4].OFF_minute; editable 0..59
rectangle at (257,129)-(478,155): tooltip Activation of the days of the week when the scheduler should be enabled
rectangle at (267,134)-(288,150): text "MO"; alarm colour if $typSchedule$.ScheduleSpecialPeriods[5].Weekday.0; toggles $typSchedule$.ScheduleSpecialPeriods[5].Weekday.0
rectangle at (297,134)-(318,150): text "TU"; alarm colour if $typSchedule$.ScheduleSpecialPeriods[5].Weekday.1; toggles $typSchedule$.ScheduleSpecialPeriods[5].Weekday.1
rectangle at (327,134)-(348,150): text "WE"; alarm colour if $typSchedule$.ScheduleSpecialPeriods[5].Weekday.2; toggles $typSchedule$.ScheduleSpecialPeriods[5].Weekday.2
rectangle at (357,134)-(378,150): text "TH"; alarm colour if $typSchedule$.ScheduleSpecialPeriods[5].Weekday.3; toggles $typSchedule$.ScheduleSpecialPeriods[5].Weekday.3
rectangle at (387,134)-(408,150): text "FR"; alarm colour if $typSchedule$.ScheduleSpecialPeriods[5].Weekday.4; toggles $typSchedule$.ScheduleSpecialPeriods[5].Weekday.4
rectangle at (417,134)-(438,150): text "SA"; alarm colour if $typSchedule$.ScheduleSpecialPeriods[5].Weekday.5; toggles $typSchedule$.ScheduleSpecialPeriods[5].Weekday.5
rectangle at (447,134)-(468,150): text "SU"; alarm colour if $typSchedule$.ScheduleSpecialPeriods[5].Weekday.6; toggles $typSchedule$.ScheduleSpecialPeriods[5].Weekday.6
rectangle at (492,134)-(508,150): alarm colour if $typSchedule$.ScheduleSpecialPeriods[5].Active.0; tooltip Indicates if time condition is fulfilled
rectangle at (167,129)-(213,155): text ":"; tooltip Switch ON time of the scheduler single period
rectangle at (172,134)-(187,150): text "%0.2d"; shows $typSchedule$.ScheduleSpecialPeriods[5].ON_hour; editable 0..23
rectangle at (193,134)-(208,150): text "%0.2d"; shows $typSchedule$.ScheduleSpecialPeriods[5].ON_minute; editable 0..59
rectangle at (87,129)-(168,155): text "_______"; tooltip Last day of the scheduler single period Input format: DD-HH-YYYY
rectangle at (93,134)-(108,150): text "%0.2d"; shows $typSchedule$.ScheduleSpecialPeriods[5].LastDay_day; editable 1..31
rectangle at (113,134)-(128,150): text "%0.2d"; shows $typSchedule$.ScheduleSpecialPeriods[5].LastDay_month; editable 1..12
rectangle at (133,134)-(163,150): text "%0.4d"; shows $typSchedule$.ScheduleSpecialPeriods[5].LastDay_year; editable 0000..2100
rectangle at (8,129)-(88,155): text "_______"; tooltip First day of the scheduler single period Input format: DD-HH-YYYY
rectangle at (33,134)-(48,150): text "%0.2d"; shows $typSchedule$.ScheduleSpecialPeriods[5].FirstDay_month; editable 1..12
rectangle at (13,134)-(28,150): text "%0.2d"; shows $typSchedule$.ScheduleSpecialPeriods[5].FirstDay_day; editable 1..31
rectangle at (53,134)-(83,150): text "%0.4d"; shows $typSchedule$.ScheduleSpecialPeriods[5].FirstDay_year; editable 0000..2100
rectangle at (212,129)-(258,155): text ":"; tooltip Switch OFF time of the scheduler single period
rectangle at (217,134)-(232,150): text "%0.2d"; shows $typSchedule$.ScheduleSpecialPeriods[5].OFF_hour; editable 0..23
rectangle at (238,134)-(253,150): text "%0.2d"; shows $typSchedule$.ScheduleSpecialPeriods[5].OFF_minute; editable 0..59
6 more shapes without text or variables
*)

(* Visualisation visuScheduler_Status
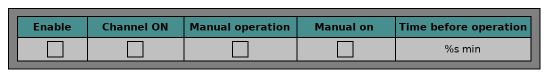
rectangle at (9,8)-(80,30): text "Enable"
rectangle at (39,33)-(55,49): alarm colour if $typSchedule$.StatusScheduler.0; tooltip Indicates if time condition is fulfilled
rectangle at (284,8)-(388,30): text "Manual on"
rectangle at (329,33)-(345,49): alarm colour if $typSchedule$.StatusScheduler.2; tooltip Indicates if time condition is fulfilled
rectangle at (175,8)-(289,30): text "Manual operation"
rectangle at (224,33)-(240,49): alarm colour if $typSchedule$.StatusScheduler.1; tooltip Indicates if time condition is fulfilled
rectangle at (387,8)-(523,30): text "Time before operation"
rectangle at (387,29)-(523,53): text "%s min"; shows $typSchedule$.TimeBeforeOperation
rectangle at (79,8)-(176,30): text "Channel ON"
rectangle at (119,33)-(135,49): alarm colour if $typSchedule$.SwitchChannel.0; tooltip Indicates if time condition is fulfilled
5 more shapes without text or variables
*)

(* Visualisation visuScheduler_Weekly
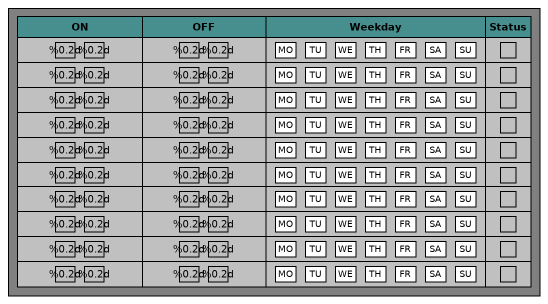
rectangle at (9,8)-(135,30): text "ON"
rectangle at (257,8)-(478,30): text "Weekday"
rectangle at (134,8)-(258,30): text "OFF"
rectangle at (477,8)-(523,30): text "Status"
rectangle at (257,29)-(478,55): tooltip Activation of the days of the week when the scheduler should be enabled
rectangle at (267,34)-(288,50): text "MO"; alarm colour if $typSchedule$.ScheduleWeekly[1].Weekday.0; toggles $typSchedule$.ScheduleWeekly[1].Weekday.0
rectangle at (297,34)-(318,50): text "TU"; alarm colour if $typSchedule$.ScheduleWeekly[1].Weekday.1; toggles $typSchedule$.ScheduleWeekly[1].Weekday.1
rectangle at (327,34)-(348,50): text "WE"; alarm colour if $typSchedule$.ScheduleWeekly[1].Weekday.2; toggles $typSchedule$.ScheduleWeekly[1].Weekday.2
rectangle at (357,34)-(378,50): text "TH"; alarm colour if $typSchedule$.ScheduleWeekly[1].Weekday.3; toggles $typSchedule$.ScheduleWeekly[1].Weekday.3
rectangle at (387,34)-(408,50): text "FR"; alarm colour if $typSchedule$.ScheduleWeekly[1].Weekday.4; toggles $typSchedule$.ScheduleWeekly[1].Weekday.4
rectangle at (417,34)-(438,50): text "SA"; alarm colour if $typSchedule$.ScheduleWeekly[1].Weekday.5; toggles $typSchedule$.ScheduleWeekly[1].Weekday.5
rectangle at (447,34)-(468,50): text "SU"; alarm colour if $typSchedule$.ScheduleWeekly[1].Weekday.6; toggles $typSchedule$.ScheduleWeekly[1].Weekday.6
rectangle at (492,34)-(508,50): alarm colour if $typSchedule$.ScheduleWeekly[1].Active.0; tooltip Indicates if time condition is fulfilled
rectangle at (9,29)-(135,55): text ":"; tooltip Switch ON time of the scheduler weekly
rectangle at (47,34)-(67,50): text "%0.2d"; shows $typSchedule$.ScheduleWeekly[1].ON_hour; editable 0..23
rectangle at (76,34)-(96,50): text "%0.2d"; shows $typSchedule$.ScheduleWeekly[1].ON_minute; editable 0..59
rectangle at (134,29)-(258,55): text ":"; tooltip Switch OFF time of the scheduler weekly
rectangle at (171,34)-(191,50): text "%0.2d"; shows $typSchedule$.ScheduleWeekly[1].OFF_hour; editable 0..23
rectangle at (200,34)-(220,50): text "%0.2d"; shows $typSchedule$.ScheduleWeekly[1].OFF_minute; editable 0..59
rectangle at (257,54)-(478,80): tooltip Activation of the days of the week when the scheduler should be enabled
rectangle at (267,59)-(288,75): text "MO"; alarm colour if $typSchedule$.ScheduleWeekly[2].Weekday.0; toggles $typSchedule$.ScheduleWeekly[2].Weekday.0
rectangle at (297,59)-(318,75): text "TU"; alarm colour if $typSchedule$.ScheduleWeekly[2].Weekday.1; toggles $typSchedule$.ScheduleWeekly[2].Weekday.1
rectangle at (327,59)-(348,75): text "WE"; alarm colour if $typSchedule$.ScheduleWeekly[2].Weekday.2; toggles $typSchedule$.ScheduleWeekly[2].Weekday.2
rectangle at (357,59)-(378,75): text "TH"; alarm colour if $typSchedule$.ScheduleWeekly[2].Weekday.3; toggles $typSchedule$.ScheduleWeekly[2].Weekday.3
rectangle at (387,59)-(408,75): text "FR"; alarm colour if $typSchedule$.ScheduleWeekly[2].Weekday.4; toggles $typSchedule$.ScheduleWeekly[2].Weekday.4
rectangle at (417,59)-(438,75): text "SA"; alarm colour if $typSchedule$.ScheduleWeekly[2].Weekday.5; toggles $typSchedule$.ScheduleWeekly[2].Weekday.5
rectangle at (447,59)-(468,75): text "SU"; alarm colour if $typSchedule$.ScheduleWeekly[2].Weekday.6; toggles $typSchedule$.ScheduleWeekly[2].Weekday.6
rectangle at (492,59)-(508,75): alarm colour if $typSchedule$.ScheduleWeekly[2].Active.0; tooltip Indicates if time condition is fulfilled
rectangle at (9,54)-(135,80): text ":"; tooltip Switch ON time of the scheduler weekly
rectangle at (47,59)-(67,75): text "%0.2d"; shows $typSchedule$.ScheduleWeekly[2].ON_hour; editable 0..23
rectangle at (76,59)-(96,75): text "%0.2d"; shows $typSchedule$.ScheduleWeekly[2].ON_minute; editable 0..59
rectangle at (134,54)-(258,80): text ":"; tooltip Switch OFF time of the scheduler weekly
rectangle at (171,59)-(191,75): text "%0.2d"; shows $typSchedule$.ScheduleWeekly[2].OFF_hour; editable 0..23
rectangle at (200,59)-(220,75): text "%0.2d"; shows $typSchedule$.ScheduleWeekly[2].OFF_minute; editable 0..59
rectangle at (257,79)-(478,105): tooltip Activation of the days of the week when the scheduler should be enabled
rectangle at (267,84)-(288,100): text "MO"; alarm colour if $typSchedule$.ScheduleWeekly[3].Weekday.0; toggles $typSchedule$.ScheduleWeekly[3].Weekday.0
rectangle at (297,84)-(318,100): text "TU"; alarm colour if $typSchedule$.ScheduleWeekly[3].Weekday.1; toggles $typSchedule$.ScheduleWeekly[3].Weekday.1
rectangle at (327,84)-(348,100): text "WE"; alarm colour if $typSchedule$.ScheduleWeekly[3].Weekday.2; toggles $typSchedule$.ScheduleWeekly[3].Weekday.2
rectangle at (357,84)-(378,100): text "TH"; alarm colour if $typSchedule$.ScheduleWeekly[3].Weekday.3; toggles $typSchedule$.ScheduleWeekly[3].Weekday.3
rectangle at (387,84)-(408,100): text "FR"; alarm colour if $typSchedule$.ScheduleWeekly[3].Weekday.4; toggles $typSchedule$.ScheduleWeekly[3].Weekday.4
rectangle at (417,84)-(438,100): text "SA"; alarm colour if $typSchedule$.ScheduleWeekly[3].Weekday.5; toggles $typSchedule$.ScheduleWeekly[3].Weekday.5
rectangle at (447,84)-(468,100): text "SU"; alarm colour if $typSchedule$.ScheduleWeekly[3].Weekday.6; toggles $typSchedule$.ScheduleWeekly[3].Weekday.6
rectangle at (492,84)-(508,100): alarm colour if $typSchedule$.ScheduleWeekly[3].Active.0; tooltip Indicates if time condition is fulfilled
rectangle at (9,79)-(135,105): text ":"; tooltip Switch ON time of the scheduler weekly
rectangle at (47,84)-(67,100): text "%0.2d"; shows $typSchedule$.ScheduleWeekly[3].ON_hour; editable 0..23
rectangle at (76,84)-(96,100): text "%0.2d"; shows $typSchedule$.ScheduleWeekly[3].ON_minute; editable 0..59
rectangle at (134,79)-(258,105): text ":"; tooltip Switch OFF time of the scheduler weekly
rectangle at (171,84)-(191,100): text "%0.2d"; shows $typSchedule$.ScheduleWeekly[3].OFF_hour; editable 0..23
rectangle at (200,84)-(220,100): text "%0.2d"; shows $typSchedule$.ScheduleWeekly[3].OFF_minute; editable 0..59
rectangle at (257,104)-(478,130): tooltip Activation of the days of the week when the scheduler should be enabled
rectangle at (267,109)-(288,125): text "MO"; alarm colour if $typSchedule$.ScheduleWeekly[4].Weekday.0; toggles $typSchedule$.ScheduleWeekly[4].Weekday.0
rectangle at (297,109)-(318,125): text "TU"; alarm colour if $typSchedule$.ScheduleWeekly[4].Weekday.1; toggles $typSchedule$.ScheduleWeekly[4].Weekday.1
rectangle at (327,109)-(348,125): text "WE"; alarm colour if $typSchedule$.ScheduleWeekly[4].Weekday.2; toggles $typSchedule$.ScheduleWeekly[4].Weekday.2
rectangle at (357,109)-(378,125): text "TH"; alarm colour if $typSchedule$.ScheduleWeekly[4].Weekday.3; toggles $typSchedule$.ScheduleWeekly[4].Weekday.3
rectangle at (387,109)-(408,125): text "FR"; alarm colour if $typSchedule$.ScheduleWeekly[4].Weekday.4; toggles $typSchedule$.ScheduleWeekly[4].Weekday.4
rectangle at (417,109)-(438,125): text "SA"; alarm colour if $typSchedule$.ScheduleWeekly[4].Weekday.5; toggles $typSchedule$.ScheduleWeekly[4].Weekday.5
rectangle at (447,109)-(468,125): text "SU"; alarm colour if $typSchedule$.ScheduleWeekly[4].Weekday.6; toggles $typSchedule$.ScheduleWeekly[4].Weekday.6
rectangle at (492,109)-(508,125): alarm colour if $typSchedule$.ScheduleWeekly[4].Active.0; tooltip Indicates if time condition is fulfilled
rectangle at (9,104)-(135,130): text ":"; tooltip Switch ON time of the scheduler weekly
rectangle at (47,109)-(67,125): text "%0.2d"; shows $typSchedule$.ScheduleWeekly[4].ON_hour; editable 0..23
rectangle at (76,109)-(96,125): text "%0.2d"; shows $typSchedule$.ScheduleWeekly[4].ON_minute; editable 0..59
rectangle at (134,104)-(258,130): text ":"; tooltip Switch OFF time of the scheduler weekly
rectangle at (171,109)-(191,125): text "%0.2d"; shows $typSchedule$.ScheduleWeekly[4].OFF_hour; editable 0..23
rectangle at (200,109)-(220,125): text "%0.2d"; shows $typSchedule$.ScheduleWeekly[4].OFF_minute; editable 0..59
rectangle at (257,129)-(478,155): tooltip Activation of the days of the week when the scheduler should be enabled
rectangle at (267,134)-(288,150): text "MO"; alarm colour if $typSchedule$.ScheduleWeekly[5].Weekday.0; toggles $typSchedule$.ScheduleWeekly[5].Weekday.0
rectangle at (297,134)-(318,150): text "TU"; alarm colour if $typSchedule$.ScheduleWeekly[5].Weekday.1; toggles $typSchedule$.ScheduleWeekly[5].Weekday.1
rectangle at (327,134)-(348,150): text "WE"; alarm colour if $typSchedule$.ScheduleWeekly[5].Weekday.2; toggles $typSchedule$.ScheduleWeekly[5].Weekday.2
rectangle at (357,134)-(378,150): text "TH"; alarm colour if $typSchedule$.ScheduleWeekly[5].Weekday.3; toggles $typSchedule$.ScheduleWeekly[5].Weekday.3
rectangle at (387,134)-(408,150): text "FR"; alarm colour if $typSchedule$.ScheduleWeekly[5].Weekday.4; toggles $typSchedule$.ScheduleWeekly[5].Weekday.4
rectangle at (417,134)-(438,150): text "SA"; alarm colour if $typSchedule$.ScheduleWeekly[5].Weekday.5; toggles $typSchedule$.ScheduleWeekly[5].Weekday.5
rectangle at (447,134)-(468,150): text "SU"; alarm colour if $typSchedule$.ScheduleWeekly[5].Weekday.6; toggles $typSchedule$.ScheduleWeekly[5].Weekday.6
rectangle at (492,134)-(508,150): alarm colour if $typSchedule$.ScheduleWeekly[5].Active.0; tooltip Indicates if time condition is fulfilled
rectangle at (9,129)-(135,155): text ":"; tooltip Switch ON time of the scheduler weekly
rectangle at (47,134)-(67,150): text "%0.2d"; shows $typSchedule$.ScheduleWeekly[5].ON_hour; editable 0..23
rectangle at (76,134)-(96,150): text "%0.2d"; shows $typSchedule$.ScheduleWeekly[5].ON_minute; editable 0..59
rectangle at (134,129)-(258,155): text ":"; tooltip Switch OFF time of the scheduler weekly
rectangle at (171,134)-(191,150): text "%0.2d"; shows $typSchedule$.ScheduleWeekly[5].OFF_hour; editable 0..23
rectangle at (200,134)-(220,150): text "%0.2d"; shows $typSchedule$.ScheduleWeekly[5].OFF_minute; editable 0..59
rectangle at (257,154)-(478,180): tooltip Activation of the days of the week when the scheduler should be enabled
rectangle at (267,159)-(288,175): text "MO"; alarm colour if $typSchedule$.ScheduleWeekly[6].Weekday.0; toggles $typSchedule$.ScheduleWeekly[6].Weekday.0
rectangle at (297,159)-(318,175): text "TU"; alarm colour if $typSchedule$.ScheduleWeekly[6].Weekday.1; toggles $typSchedule$.ScheduleWeekly[6].Weekday.1
rectangle at (327,159)-(348,175): text "WE"; alarm colour if $typSchedule$.ScheduleWeekly[6].Weekday.2; toggles $typSchedule$.ScheduleWeekly[6].Weekday.2
rectangle at (357,159)-(378,175): text "TH"; alarm colour if $typSchedule$.ScheduleWeekly[6].Weekday.3; toggles $typSchedule$.ScheduleWeekly[6].Weekday.3
rectangle at (387,159)-(408,175): text "FR"; alarm colour if $typSchedule$.ScheduleWeekly[6].Weekday.4; toggles $typSchedule$.ScheduleWeekly[6].Weekday.4
rectangle at (417,159)-(438,175): text "SA"; alarm colour if $typSchedule$.ScheduleWeekly[6].Weekday.5; toggles $typSchedule$.ScheduleWeekly[6].Weekday.5
rectangle at (447,159)-(468,175): text "SU"; alarm colour if $typSchedule$.ScheduleWeekly[6].Weekday.6; toggles $typSchedule$.ScheduleWeekly[6].Weekday.6
rectangle at (492,159)-(508,175): alarm colour if $typSchedule$.ScheduleWeekly[6].Active.0; tooltip Indicates if time condition is fulfilled
rectangle at (9,154)-(135,180): text ":"; tooltip Switch ON time of the scheduler weekly
rectangle at (47,159)-(67,175): text "%0.2d"; shows $typSchedule$.ScheduleWeekly[6].ON_hour; editable 0..23
rectangle at (76,159)-(96,175): text "%0.2d"; shows $typSchedule$.ScheduleWeekly[6].ON_minute; editable 0..59
rectangle at (134,154)-(258,180): text ":"; tooltip Switch OFF time of the scheduler weekly
rectangle at (171,159)-(191,175): text "%0.2d"; shows $typSchedule$.ScheduleWeekly[6].OFF_hour; editable 0..23
rectangle at (200,159)-(220,175): text "%0.2d"; shows $typSchedule$.ScheduleWeekly[6].OFF_minute; editable 0..59
rectangle at (257,178)-(478,204): tooltip Activation of the days of the week when the scheduler should be enabled
rectangle at (267,183)-(288,199): text "MO"; alarm colour if $typSchedule$.ScheduleWeekly[7].Weekday.0; toggles $typSchedule$.ScheduleWeekly[7].Weekday.0
rectangle at (297,183)-(318,199): text "TU"; alarm colour if $typSchedule$.ScheduleWeekly[7].Weekday.1; toggles $typSchedule$.ScheduleWeekly[7].Weekday.1
rectangle at (327,183)-(348,199): text "WE"; alarm colour if $typSchedule$.ScheduleWeekly[7].Weekday.2; toggles $typSchedule$.ScheduleWeekly[7].Weekday.2
rectangle at (357,183)-(378,199): text "TH"; alarm colour if $typSchedule$.ScheduleWeekly[7].Weekday.3; toggles $typSchedule$.ScheduleWeekly[7].Weekday.3
rectangle at (387,183)-(408,199): text "FR"; alarm colour if $typSchedule$.ScheduleWeekly[7].Weekday.4; toggles $typSchedule$.ScheduleWeekly[7].Weekday.4
rectangle at (417,183)-(438,199): text "SA"; alarm colour if $typSchedule$.ScheduleWeekly[7].Weekday.5; toggles $typSchedule$.ScheduleWeekly[7].Weekday.5
rectangle at (447,183)-(468,199): text "SU"; alarm colour if $typSchedule$.ScheduleWeekly[7].Weekday.6; toggles $typSchedule$.ScheduleWeekly[7].Weekday.6
rectangle at (492,183)-(508,199): alarm colour if $typSchedule$.ScheduleWeekly[7].Active.0; tooltip Indicates if time condition is fulfilled
rectangle at (9,178)-(135,204): text ":"; tooltip Switch ON time of the scheduler weekly
rectangle at (47,183)-(67,199): text "%0.2d"; shows $typSchedule$.ScheduleWeekly[7].ON_hour; editable 0..23
rectangle at (76,183)-(96,199): text "%0.2d"; shows $typSchedule$.ScheduleWeekly[7].ON_minute; editable 0..59
rectangle at (134,178)-(258,204): text ":"; tooltip Switch OFF time of the scheduler weekly
rectangle at (171,183)-(191,199): text "%0.2d"; shows $typSchedule$.ScheduleWeekly[7].OFF_hour; editable 0..23
rectangle at (200,183)-(220,199): text "%0.2d"; shows $typSchedule$.ScheduleWeekly[7].OFF_minute; editable 0..59
rectangle at (257,203)-(478,229): tooltip Activation of the days of the week when the scheduler should be enabled
rectangle at (267,208)-(288,224): text "MO"; alarm colour if $typSchedule$.ScheduleWeekly[8].Weekday.0; toggles $typSchedule$.ScheduleWeekly[8].Weekday.0
rectangle at (297,208)-(318,224): text "TU"; alarm colour if $typSchedule$.ScheduleWeekly[8].Weekday.1; toggles $typSchedule$.ScheduleWeekly[8].Weekday.1
rectangle at (327,208)-(348,224): text "WE"; alarm colour if $typSchedule$.ScheduleWeekly[8].Weekday.2; toggles $typSchedule$.ScheduleWeekly[8].Weekday.2
rectangle at (357,208)-(378,224): text "TH"; alarm colour if $typSchedule$.ScheduleWeekly[8].Weekday.3; toggles $typSchedule$.ScheduleWeekly[8].Weekday.3
rectangle at (387,208)-(408,224): text "FR"; alarm colour if $typSchedule$.ScheduleWeekly[8].Weekday.4; toggles $typSchedule$.ScheduleWeekly[8].Weekday.4
rectangle at (417,208)-(438,224): text "SA"; alarm colour if $typSchedule$.ScheduleWeekly[8].Weekday.5; toggles $typSchedule$.ScheduleWeekly[8].Weekday.5
rectangle at (447,208)-(468,224): text "SU"; alarm colour if $typSchedule$.ScheduleWeekly[8].Weekday.6; toggles $typSchedule$.ScheduleWeekly[8].Weekday.6
rectangle at (492,208)-(508,224): alarm colour if $typSchedule$.ScheduleWeekly[8].Active.0; tooltip Indicates if time condition is fulfilled
rectangle at (9,203)-(135,229): text ":"; tooltip Switch ON time of the scheduler weekly
rectangle at (47,208)-(67,224): text "%0.2d"; shows $typSchedule$.ScheduleWeekly[8].ON_hour; editable 0..23
rectangle at (76,208)-(96,224): text "%0.2d"; shows $typSchedule$.ScheduleWeekly[8].ON_minute; editable 0..59
rectangle at (134,203)-(258,229): text ":"; tooltip Switch OFF time of the scheduler weekly
rectangle at (171,208)-(191,224): text "%0.2d"; shows $typSchedule$.ScheduleWeekly[8].OFF_hour; editable 0..23
rectangle at (200,208)-(220,224): text "%0.2d"; shows $typSchedule$.ScheduleWeekly[8].OFF_minute; editable 0..59
rectangle at (257,228)-(478,254): tooltip Activation of the days of the week when the scheduler should be enabled
rectangle at (267,233)-(288,249): text "MO"; alarm colour if $typSchedule$.ScheduleWeekly[9].Weekday.0; toggles $typSchedule$.ScheduleWeekly[9].Weekday.0
rectangle at (297,233)-(318,249): text "TU"; alarm colour if $typSchedule$.ScheduleWeekly[9].Weekday.1; toggles $typSchedule$.ScheduleWeekly[9].Weekday.1
rectangle at (327,233)-(348,249): text "WE"; alarm colour if $typSchedule$.ScheduleWeekly[9].Weekday.2; toggles $typSchedule$.ScheduleWeekly[9].Weekday.2
rectangle at (357,233)-(378,249): text "TH"; alarm colour if $typSchedule$.ScheduleWeekly[9].Weekday.3; toggles $typSchedule$.ScheduleWeekly[9].Weekday.3
rectangle at (387,233)-(408,249): text "FR"; alarm colour if $typSchedule$.ScheduleWeekly[9].Weekday.4; toggles $typSchedule$.ScheduleWeekly[9].Weekday.4
rectangle at (417,233)-(438,249): text "SA"; alarm colour if $typSchedule$.ScheduleWeekly[9].Weekday.5; toggles $typSchedule$.ScheduleWeekly[9].Weekday.5
rectangle at (447,233)-(468,249): text "SU"; alarm colour if $typSchedule$.ScheduleWeekly[9].Weekday.6; toggles $typSchedule$.ScheduleWeekly[9].Weekday.6
rectangle at (492,233)-(508,249): alarm colour if $typSchedule$.ScheduleWeekly[9].Active.0; tooltip Indicates if time condition is fulfilled
rectangle at (9,228)-(135,254): text ":"; tooltip Switch ON time of the scheduler weekly
rectangle at (47,233)-(67,249): text "%0.2d"; shows $typSchedule$.ScheduleWeekly[9].ON_hour; editable 0..23
rectangle at (76,233)-(96,249): text "%0.2d"; shows $typSchedule$.ScheduleWeekly[9].ON_minute; editable 0..59
rectangle at (134,228)-(258,254): text ":"; tooltip Switch OFF time of the scheduler weekly
rectangle at (171,233)-(191,249): text "%0.2d"; shows $typSchedule$.ScheduleWeekly[9].OFF_hour; editable 0..23
rectangle at (200,233)-(220,249): text "%0.2d"; shows $typSchedule$.ScheduleWeekly[9].OFF_minute; editable 0..59
rectangle at (257,253)-(478,279): tooltip Activation of the days of the week when the scheduler should be enabled
rectangle at (267,258)-(288,274): text "MO"; alarm colour if $typSchedule$.ScheduleWeekly[10].Weekday.0; toggles $typSchedule$.ScheduleWeekly[10].Weekday.0
rectangle at (297,258)-(318,274): text "TU"; alarm colour if $typSchedule$.ScheduleWeekly[10].Weekday.1; toggles $typSchedule$.ScheduleWeekly[10].Weekday.1
rectangle at (327,258)-(348,274): text "WE"; alarm colour if $typSchedule$.ScheduleWeekly[10].Weekday.2; toggles $typSchedule$.ScheduleWeekly[10].Weekday.2
rectangle at (357,258)-(378,274): text "TH"; alarm colour if $typSchedule$.ScheduleWeekly[10].Weekday.3; toggles $typSchedule$.ScheduleWeekly[10].Weekday.3
rectangle at (387,258)-(408,274): text "FR"; alarm colour if $typSchedule$.ScheduleWeekly[10].Weekday.4; toggles $typSchedule$.ScheduleWeekly[10].Weekday.4
rectangle at (417,258)-(438,274): text "SA"; alarm colour if $typSchedule$.ScheduleWeekly[10].Weekday.5; toggles $typSchedule$.ScheduleWeekly[10].Weekday.5
rectangle at (447,258)-(468,274): text "SU"; alarm colour if $typSchedule$.ScheduleWeekly[10].Weekday.6; toggles $typSchedule$.ScheduleWeekly[10].Weekday.6
rectangle at (492,258)-(508,274): alarm colour if $typSchedule$.ScheduleWeekly[10].Active.0; tooltip Indicates if time condition is fulfilled
rectangle at (9,253)-(135,279): text ":"; tooltip Switch ON time of the scheduler weekly
rectangle at (47,258)-(67,274): text "%0.2d"; shows $typSchedule$.ScheduleWeekly[10].ON_hour; editable 0..23
rectangle at (76,258)-(96,274): text "%0.2d"; shows $typSchedule$.ScheduleWeekly[10].ON_minute; editable 0..59
rectangle at (134,253)-(258,279): text ":"; tooltip Switch OFF time of the scheduler weekly
rectangle at (171,258)-(191,274): text "%0.2d"; shows $typSchedule$.ScheduleWeekly[10].OFF_hour; editable 0..23
rectangle at (200,258)-(220,274): text "%0.2d"; shows $typSchedule$.ScheduleWeekly[10].OFF_minute; editable 0..59
11 more shapes without text or variables
*)

(* Visualisation visuScheduleSpecialPeriod
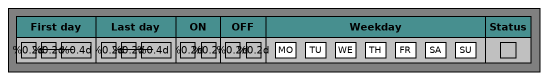
rectangle at (167,8)-(213,30): text "ON"
rectangle at (257,8)-(478,30): text "Weekday"
rectangle at (212,8)-(258,30): text "OFF"
rectangle at (87,8)-(168,30): text "Last day"
rectangle at (8,8)-(88,30): text "First day"
rectangle at (477,8)-(523,30): text "Status"
rectangle at (257,29)-(478,55): tooltip Activation of the days of the week when the scheduler should be enabled
rectangle at (267,34)-(288,50): text "MO"; alarm colour if $typScheduleSpecialPeriod$.Weekday.0; toggles $typScheduleSpecialPeriod$.Weekday.0
rectangle at (297,34)-(318,50): text "TU"; alarm colour if $typScheduleSpecialPeriod$.Weekday.1; toggles $typScheduleSpecialPeriod$.Weekday.1
rectangle at (327,34)-(348,50): text "WE"; alarm colour if $typScheduleSpecialPeriod$.Weekday.2; toggles $typScheduleSpecialPeriod$.Weekday.2
rectangle at (357,34)-(378,50): text "TH"; alarm colour if $typScheduleSpecialPeriod$.Weekday.3; toggles $typScheduleSpecialPeriod$.Weekday.3
rectangle at (387,34)-(408,50): text "FR"; alarm colour if $typScheduleSpecialPeriod$.Weekday.4; toggles $typScheduleSpecialPeriod$.Weekday.4
rectangle at (417,34)-(438,50): text "SA"; alarm colour if $typScheduleSpecialPeriod$.Weekday.5; toggles $typScheduleSpecialPeriod$.Weekday.5
rectangle at (447,34)-(468,50): text "SU"; alarm colour if $typScheduleSpecialPeriod$.Weekday.6; toggles $typScheduleSpecialPeriod$.Weekday.6
rectangle at (492,34)-(508,50): alarm colour if $typScheduleSpecialPeriod$.Active.0; tooltip Indicates if time condition is fulfilled
rectangle at (167,29)-(213,55): text ":"; tooltip Switch ON time of the scheduler single period
rectangle at (172,34)-(187,50): text "%0.2d"; shows $typScheduleSpecialPeriod$.ON_hour; editable 0..23
rectangle at (193,34)-(208,50): text "%0.2d"; shows $typScheduleSpecialPeriod$.ON_minute; editable 0..59
rectangle at (87,29)-(168,55): text "_______"; tooltip Last day of the scheduler single period Input format: DD-HH-YYYY
rectangle at (93,34)-(108,50): text "%0.2d"; shows $typScheduleSpecialPeriod$.LastDay_day; editable 1..31
rectangle at (113,34)-(128,50): text "%0.2d"; shows $typScheduleSpecialPeriod$.LastDay_month; editable 1..12
rectangle at (133,34)-(163,50): text "%0.4d"; shows $typScheduleSpecialPeriod$.LastDay_year; editable 0000..2100
rectangle at (8,29)-(88,55): text "_______"; tooltip First day of the scheduler single period Input format: DD-HH-YYYY
rectangle at (33,34)-(48,50): text "%0.2d"; shows $typScheduleSpecialPeriod$.FirstDay_month; editable 1..12
rectangle at (13,34)-(28,50): text "%0.2d"; shows $typScheduleSpecialPeriod$.FirstDay_day; editable 1..31
rectangle at (53,34)-(83,50): text "%0.4d"; shows $typScheduleSpecialPeriod$.FirstDay_year; editable 0000..2100
rectangle at (212,29)-(258,55): text ":"; tooltip Switch OFF time of the scheduler single period
rectangle at (217,34)-(232,50): text "%0.2d"; shows $typScheduleSpecialPeriod$.OFF_hour; editable 0..23
rectangle at (238,34)-(253,50): text "%0.2d"; shows $typScheduleSpecialPeriod$.OFF_minute; editable 0..59
2 more shapes without text or variables
*)

(* Visualisation visuScheduleWeekly
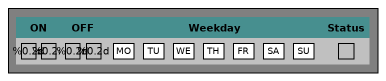
rectangle at (8,30)-(361,56): tooltip Activation of the days of the week when the scheduler should be enabled
rectangle at (97,9)-(316,31): text "Weekday"
rectangle at (8,9)-(53,31): text "ON"
rectangle at (52,9)-(98,31): text "OFF"
rectangle at (315,9)-(361,31): text "Status"
rectangle at (97,30)-(316,56): tooltip Activation of the days of the week when the scheduler should be enabled
rectangle at (105,35)-(126,51): text "MO"; alarm colour if $typScheduleWeekly$.Weekday.0; toggles $typScheduleWeekly$.Weekday.0
rectangle at (135,35)-(156,51): text "TU"; alarm colour if $typScheduleWeekly$.Weekday.1; toggles $typScheduleWeekly$.Weekday.1
rectangle at (165,35)-(186,51): text "WE"; alarm colour if $typScheduleWeekly$.Weekday.2; toggles $typScheduleWeekly$.Weekday.2
rectangle at (195,35)-(216,51): text "TH"; alarm colour if $typScheduleWeekly$.Weekday.3; toggles $typScheduleWeekly$.Weekday.3
rectangle at (225,35)-(246,51): text "FR"; alarm colour if $typScheduleWeekly$.Weekday.4; toggles $typScheduleWeekly$.Weekday.4
rectangle at (255,35)-(276,51): text "SA"; alarm colour if $typScheduleWeekly$.Weekday.5; toggles $typScheduleWeekly$.Weekday.5
rectangle at (285,35)-(306,51): text "SU"; alarm colour if $typScheduleWeekly$.Weekday.6; toggles $typScheduleWeekly$.Weekday.6
rectangle at (330,35)-(346,51): alarm colour if $typScheduleWeekly$.Active.0; tooltip Indicates if time condition is fulfilled
rectangle at (8,30)-(53,56): text ":"; tooltip Switch ON time of the scheduler single weekly
rectangle at (13,35)-(28,51): text "%0.2d"; shows $typScheduleWeekly$.ON_hour; editable 0..23
rectangle at (33,35)-(48,51): text "%0.2d"; shows $typScheduleWeekly$.ON_minute; editable 0..59
rectangle at (52,30)-(98,56): text ":"; tooltip Switch OFF time of the scheduler single weekly
rectangle at (57,35)-(72,51): text "%0.2d"; shows $typScheduleWeekly$.OFF_hour; editable 0..23
rectangle at (78,35)-(93,51): text "%0.2d"; shows $typScheduleWeekly$.OFF_minute; editable 0..59
3 more shapes without text or variables
*)

(* Visualisation visuSetScheduleValue_SpecialPeriods
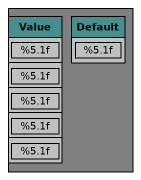
rectangle at (0,8)-(54,30): text "Value"
rectangle at (0,29)-(54,55): tooltip Value of the scheduler SpecialPeriods
rectangle at (3,34)-(51,50): text "%5.1f"; shows $typScheduleValue$.arSpecial[1]; editable
rectangle at (0,54)-(54,80): tooltip Value of the scheduler SpecialPeriods
rectangle at (0,79)-(54,105): tooltip Value of the scheduler SpecialPeriods
rectangle at (0,104)-(54,130): tooltip Value of the scheduler SpecialPeriods
rectangle at (0,129)-(54,155): tooltip Value of the scheduler SpecialPeriods
rectangle at (3,60)-(51,76): text "%5.1f"; shows $typScheduleValue$.arSpecial[2]; editable
rectangle at (3,85)-(51,101): text "%5.1f"; shows $typScheduleValue$.arSpecial[3]; editable
rectangle at (3,110)-(51,126): text "%5.1f"; shows $typScheduleValue$.arSpecial[4]; editable
rectangle at (3,135)-(51,151): text "%5.1f"; shows $typScheduleValue$.arSpecial[5]; editable
rectangle at (63,8)-(117,30): text "Default"
rectangle at (63,29)-(117,55): tooltip Default-Value of the scheduler
rectangle at (67,34)-(113,50): text "%5.1f"; shows $typScheduleValue$.rDefault; editable
1 more shapes without text or variables
*)

(* Visualisation visuSetScheduleValue_Weekly
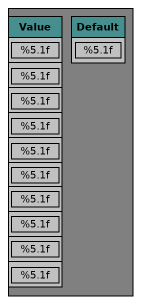
rectangle at (-1,8)-(53,30): text "Value"
rectangle at (-1,29)-(53,55): tooltip Value of the scheduler weekly
rectangle at (2,34)-(50,50): text "%5.1f"; shows $typScheduleValue$.arWeekly[1]; editable
rectangle at (-1,54)-(53,80): tooltip Value of the scheduler weekly
rectangle at (-1,79)-(53,105): tooltip Value of the scheduler weekly
rectangle at (-1,104)-(53,130): tooltip Value of the scheduler weekly
rectangle at (-1,129)-(53,155): tooltip Value of the scheduler weekly
rectangle at (-1,154)-(53,180): tooltip Value of the scheduler weekly
rectangle at (-1,178)-(53,204): tooltip Value of the scheduler weekly
rectangle at (-1,203)-(53,229): tooltip Value of the scheduler weekly
rectangle at (-1,228)-(53,254): tooltip Value of the scheduler weekly
rectangle at (-1,253)-(53,279): tooltip Value of the scheduler weekly
rectangle at (2,60)-(50,76): text "%5.1f"; shows $typScheduleValue$.arWeekly[2]; editable
rectangle at (2,85)-(50,101): text "%5.1f"; shows $typScheduleValue$.arWeekly[3]; editable
rectangle at (2,110)-(50,126): text "%5.1f"; shows $typScheduleValue$.arWeekly[4]; editable
rectangle at (2,135)-(50,151): text "%5.1f"; shows $typScheduleValue$.arWeekly[5]; editable
rectangle at (2,159)-(50,175): text "%5.1f"; shows $typScheduleValue$.arWeekly[6]; editable
rectangle at (2,183)-(50,199): text "%5.1f"; shows $typScheduleValue$.arWeekly[7]; editable
rectangle at (2,208)-(50,224): text "%5.1f"; shows $typScheduleValue$.arWeekly[8]; editable
rectangle at (2,233)-(50,249): text "%5.1f"; shows $typScheduleValue$.arWeekly[9]; editable
rectangle at (2,259)-(50,275): text "%5.1f"; shows $typScheduleValue$.arWeekly[10]; editable
rectangle at (62,8)-(116,30): text "Default"
rectangle at (62,29)-(116,55): tooltip Default-Value of the scheduler
rectangle at (66,34)-(112,50): text "%5.1f"; shows $typScheduleValue$.rDefault; editable
1 more shapes without text or variables
*)

